TYPE "SpeedMachine_CIn_Manager"
VERSION : 0.1
// Block: SpeedMachine_CIn_Manager
   STRUCT
      EnableStopDoorOpeningReq : Bool;
      EnableStopInPhase : Bool;
      EnableStopProgrammed : Bool;
      Control_ON : Bool;
      Bwd : Bool;
      Fwd : Bool;
      Vel : LReal;
      Acc : LReal;
      Dec : LReal;
   END_STRUCT;

END_TYPE
